TYPE stAxisInterface :
STRUCT
	

IN	:	stAxisIN;
OUT	:	stAxisOUT;


END_STRUCT
END_TYPE

(* stored: Version 1.1.0.1, ProductVersion 3.1.4024.4
   DUT stAxisInterface: Id {08153def-bc3a-491b-b5c5-54661bb763b9} *)
